// TIA Portal V20 export
FUNCTION "StepToString" : String   // FC87, SCL
// stored: Namespace Unit1.Em7, SetENOAutomatically false
   VAR_INPUT
      StepDINT : DInt;   // DINT value of the step
   END_VAR
BEGIN
   // Translates shared conveyor sequence step numbers to step names
   // Sequence-specific duplicate numbers are expressed as combined labels

   CASE #StepDINT OF
       1:
           #StepToString := 'Idle';

       101:
           #StepToString := 'JOB[1] Condition';
       111:
           #StepToString := 'RingBlow / Kicker / Stack QR Ready Check';
       121:
           #StepToString := 'Conveyor Homed / Kicker HomePos Check';
       131:
           #StepToString := 'NG Box Lock Cylinder WorkPos Check';
       191:
           #StepToString := 'JOB[1] Step End';

       201:
           #StepToString := 'JOB[2] Condition';
       211:
           #StepToString := 'Spare / Kicker Move / QR Trigger / Load Request';
       221:
           #StepToString := 'Load Enable On';
       231:
           #StepToString := 'Cell Data Report';
       241:
           #StepToString := 'Load Enable Off';
       251:
           #StepToString := 'Load Complete';
       291:
           #StepToString := 'JOB[2] Step End';

       301:
           #StepToString := 'JOB[3] Condition';
       311:
           #StepToString := 'Conveyor GearIn Command';
       321:
           #StepToString := 'Conveyor Virtual Axis posRelative Command';
       391:
           #StepToString := 'JOB[3] Step End';

       801:
           #StepToString := 'JOB[8] Condition';
       811:
           #StepToString := 'Manual P&P Unloading Request';
       821:
           #StepToString := 'Manual P&P Unloading Done';
       891:
           #StepToString := 'JOB[8] Step End';

       901:
           #StepToString := 'JOB[9] Condition / Immediate Stop';
       911:
           #StepToString := 'Vision Inspection Request';
       921:
           #StepToString := 'Vision Inspection Done';
       991:
           #StepToString := 'JOB[9] Step End';

       1001:
           #StepToString := 'JOB[10] Condition';
       1011:
           #StepToString := 'Cut Conveyor Axis B Move FWD';
       1021:
           #StepToString := 'Vision Inspection Request';
       1031:
           #StepToString := 'Vision Inspection Done';
       1041:
           #StepToString := 'Cut Conveyor Axis B Move BWD';
       1091:
           #StepToString := 'JOB[10] Step End';

       9001:
           #StepToString := 'Immediate Stop';

       ELSE
           #StepToString := 'N/A';

   END_CASE;
END_FUNCTION
